(* IEC 61131-3 sources: ATCMcontrol_Engineering/src/TargetBase/Libs/ATCM_IEC1131_3/table_27, 5 files *)

(* ---- limit.st ---- *)
(*[[
    UserURL= "ATCMfile:LIMIT.htm"
]]*)

FUNCTION LIMIT : ANY_ELEMENTARY
VAR_INPUT
    MN : ANY_ELEMENTARY;
    IN : ANY_ELEMENTARY;
    MX : ANY_ELEMENTARY;
END_VAR

overload BOOL(BOOL,BOOL,BOOL) inline
{
    %2
    %1
    or_bool
    %3
    and_bool
}
overload BYTE(BYTE, BYTE, BYTE) inline
{
    %2
    %1
    lt_byte
    jmpcn L1%u
    %1
    jmp Lend%u
:L1%u
    %2
    %3
    gt_byte
    jmpcn L2%u
    %3
    jmp Lend%u
:L2%u
    %2
:Lend%u
}
overload WORD(WORD, WORD, WORD) inline
{
    %2
    %1
    lt_word
    jmpcn L1%u
    %1
    jmp Lend%u
:L1%u
    %2
    %3
    gt_word
    jmpcn L2%u
    %3
    jmp Lend%u
:L2%u
    %2
:Lend%u
}
overload DWORD(DWORD, DWORD, DWORD) inline
{
    %2
    %1
    lt_dword
    jmpcn L1%u
    %1
    jmp Lend%u
:L1%u
    %2
    %3
    gt_dword
    jmpcn L2%u
    %3
    jmp Lend%u
:L2%u
    %2
:Lend%u
}
overload INT(INT, INT, INT) inline
{
    %2
    %1
    lt_int
    jmpcn L1%u
    %1
    jmp Lend%u
:L1%u
    %2
    %3
    gt_int
    jmpcn L2%u
    %3
    jmp Lend%u
:L2%u
    %2
:Lend%u
}
overload DINT|TIME(DINT|TIME, DINT|TIME, DINT|TIME) inline
{
    %2
    %1
    lt_dint
    jmpcn L1%u
    %1
    jmp Lend%u
:L1%u
    %2
    %3
    gt_dint
    jmpcn L2%u
    %3
    jmp Lend%u
:L2%u
    %2
:Lend%u
}
overload REAL(REAL,REAL,REAL) inline
{
    %2
    %1
    lt_real
    jmpcn L1%u
    %1
    jmp Lend%u
:L1%u
    %2
    %3
    gt_real
    jmpcn L2%u
    %3
    jmp Lend%u
:L2%u
    %2
:Lend%u
}

overload LREAL(LREAL,LREAL,LREAL) inline
{
    %2
    %1
    lt_lreal
    jmpcn L1%u
    %1
    jmp Lend%u
:L1%u
    %2
    %3
    gt_lreal
    jmpcn L2%u
    %3
    jmp Lend%u
:L2%u
    %2
:Lend%u
}

overload STRING(STRING, STRING, STRING) inline
{
    %2
    %1
    lt_string
    jmpcn L1%u
    %1
    jmp Lend%u
:L1%u
    %2
    %3
    gt_string
    jmpcn L2%u
    %3
    jmp Lend%u
:L2%u
    %2
:Lend%u
}

END_FUNCTION

(* ---- max.st ---- *)
(*[[
]]*)

FUNCTION MAX : ANY_ELEMENTARY
VAR_INPUT
    IN1 : ANY_ELEMENTARY;
END_VAR
VAR_IN_EXT
    IN2 : ANY_ELEMENTARY;
END_VAR

overload BOOL(BOOL,BOOL) inline
{
    %1
    %2
    or_bool
}
overload BYTE(BYTE,BYTE) inline
{
    %1
    %2
    gt_byte
    jmpcn L1%u
    %1
    jmp Lend%u
:L1%u
    %2
:Lend%u
}
overload WORD(WORD,WORD) inline
{
    %1
    %2
    gt_word
    jmpcn L1%u
    %1
    jmp Lend%u
:L1%u
    %2
:Lend%u
}
overload DWORD(DWORD,DWORD) inline
{
    %1
    %2
    gt_dword
    jmpcn L1%u
    %1
    jmp Lend%u
:L1%u
    %2
:Lend%u
}
overload INT(INT,INT) inline
{
    %1
    %2
    gt_int
    jmpcn L1%u
    %1
    jmp Lend%u
:L1%u
    %2
:Lend%u
}
overload DINT|TIME(DINT|TIME,DINT|TIME) inline
{
    %1
    %2
    gt_dint
    jmpcn L1%u
    %1
    jmp Lend%u
:L1%u
    %2
:Lend%u
}
overload REAL(REAL,REAL) inline
{
    %1
    %2
    gt_real
    jmpcn L1%u
    %1
    jmp Lend%u
:L1%u
    %2
:Lend%u
}
overload LREAL(LREAL,LREAL) inline
{
    %1
    %2
    gt_lreal
    jmpcn L1%u
    %1
    jmp Lend%u
:L1%u
    %2
:Lend%u
}
overload STRING(STRING,STRING) inline
{
    %1
    %2
    gt_string
    jmpcn L1%u
    %1
    jmp Lend%u
:L1%u
    %2
:Lend%u
}

(*
TODO implement extensible funs in interpreter
overload BOOL(BOOL, BOOL, ... )                        inline{ STDLIB(max_bool) }
overload BYTE(BYTE,BYTE, ... )                         inline{ STDLIB(max_byte) }
overload WORD(WORD,WORD, ... )                         inline{ STDLIB(max_word) }
overload DWORD(DWORD, DWORD, ... )                     inline{ STDLIB(max_dword) }

overload INT(INT,INT, ... )                            inline{ STDLIB(max_int) }
overload DINT(DINT,DINT, ... )                         inline{ STDLIB(max_dint) }

overload REAL(REAL,REAL, ... )                         inline{ STDLIB(max_real) }
overload LREAL(LREAL,LREAL, ... )                      inline{ STDLIB(max_lreal) }

overload TIME(TIME,TIME, ...)                          inline{ STDLIB(max_udint) }
overload STRING(STRING, STRING, ... )                  inline{ STDLIB(max_string) }
*)

END_FUNCTION

(* ---- MIN.st ---- *)
FUNCTION MIN : ANY_ELEMENTARY
VAR_INPUT
    IN1 : ANY_ELEMENTARY;
END_VAR
VAR_IN_EXT
    IN2 : ANY_ELEMENTARY;
END_VAR

overload BOOL(BOOL,BOOL) inline
{
    %1
    %2
    and_bool
}
overload BYTE(BYTE,BYTE) inline
{
    %1
    %2
    lt_byte
    jmpcn L1%u
    %1
    jmp Lend%u
:L1%u
    %2
:Lend%u
}
overload WORD(WORD,WORD) inline
{
    %1
    %2
    lt_word
    jmpcn L1%u
    %1
    jmp Lend%u
:L1%u
    %2
:Lend%u
}
overload DWORD(DWORD,DWORD) inline
{
    %1
    %2
    lt_dword
    jmpcn L1%u
    %1
    jmp Lend%u
:L1%u
    %2
:Lend%u
}
overload INT(INT,INT) inline
{
    %1
    %2
    lt_int
    jmpcn L1%u
    %1
    jmp Lend%u
:L1%u
    %2
:Lend%u
}
overload DINT|TIME(DINT|TIME,DINT|TIME) inline
{
    %1
    %2
    lt_dint
    jmpcn L1%u
    %1
    jmp Lend%u
:L1%u
    %2
:Lend%u
}
overload REAL(REAL,REAL) inline
{
    %1
    %2
    lt_real
    jmpcn L1%u
    %1
    jmp Lend%u
:L1%u
    %2
:Lend%u
}
overload LREAL(LREAL,LREAL) inline
{
    %1
    %2
    lt_lreal
    jmpcn L1%u
    %1
    jmp Lend%u
:L1%u
    %2
:Lend%u
}

overload STRING(STRING,STRING) inline
{
    %1
    %2
    lt_string
    jmpcn L1%u
    %1
    jmp Lend%u
:L1%u
    %2
:Lend%u
}

(*
TODO implement extensible funs in interpreter
overload BOOL(BOOL, BOOL, ... )                        inline{ STDLIB(min_bool) }
overload BYTE(BYTE,BYTE, ... )                         inline{ STDLIB(min_byte) }
overload WORD(WORD,WORD, ... )                         inline{ STDLIB(min_word) }
overload DWORD(DWORD, DWORD, ... )                     inline{ STDLIB(min_dword) }

overload INT(INT,INT, ... )                            inline{ STDLIB(min_int) }
overload DINT(DINT,DINT, ... )                         inline{ STDLIB(min_dint) }

overload REAL(REAL,REAL, ... )                         inline{ STDLIB(min_real) }
overload LREAL(LREAL,LREAL, ... )                      inline{ STDLIB(min_lreal) }

overload TIME(TIME,TIME, ...)                          inline{ STDLIB(min_udint) }
overload STRING(STRING, STRING, ... )                  inline{ STDLIB(min_string) }
*)

END_FUNCTION

(* ---- MUX.st ---- *)
FUNCTION MUX : ANY
VAR_INPUT
   K : ANY_INT;
   IN0: ANY;
END_VAR
VAR_IN_EXT
   IN1: ANY;
END_VAR

(* 1 bit *)
overload BOOL  (INT|DINT to INT, BOOL,   ...) inline{ STDLIB(mux_bit) }

(* 8 bit *)
overload BYTE  (INT|DINT to INT, BYTE,   ...) inline{ STDLIB(mux_byte) }

(* 16 bit *)
overload INT   (INT|DINT to INT, INT,    ...) inline{ STDLIB(mux_int) }
overload WORD  (INT|DINT to INT, WORD,   ...) inline{ STDLIB(mux_int) }

(* 32 bit *)
overload DINT  (INT|DINT to INT, DINT,   ...) inline{ STDLIB(mux_dint) }
overload DWORD (INT|DINT to INT, DWORD,  ...) inline{ STDLIB(mux_dint) }
overload TIME  (INT|DINT to INT, TIME,   ...) inline{ STDLIB(mux_dint) }
overload REAL  (INT|DINT to INT, REAL,   ...) inline{ STDLIB(mux_dint) }

(* 64 bit *)
overload LREAL (INT|DINT to INT, LREAL,  ...) inline{ STDLIB(mux_64bit) }

(* string *)
overload STRING(INT|DINT to INT, STRING, ...) inline{ STDLIB(mux_string) }

END_FUNCTION

(* ---- SEL.st ---- *)
FUNCTION SEL : ANY

VAR_INPUT
    G   : BOOL;
    IN0 : ANY;
    IN1 : ANY;
END_VAR

overload ANY_ELEMENTARY(BOOL,ANY_ELEMENTARY,ANY_ELEMENTARY) inline
{
    %1
    jmpcn L1%u
    %3
    jmp L2%u
:L1%u
    %2
:L2%u
}
END_FUNCTION
